FUNCTION_BLOCK DataManager EXTENDS TcoData.TcoDataExchange
VAR
	_data : Data;
END_VAR

SUPER^();

END_FUNCTION_BLOCK

(* stored: Version 1.1.0.1, ProductVersion 3.1.4024.9
   POU DataManager: Id {2fa16878-1e00-032b-0e94-c02db7ea7b02}, SpecialFunc None *)
